(* CODESYS project ObjectOrientedProgramming(Extended).project
   Description: This example demonstrates how object orientation is used to realize a building with different rooms, which have different functions. The included visualization illustrates the implementation.
   Title: Extended Example for Object Oriented Programming

Project tree, tasks and I/O mapping:
  Device : CODESYS Control Win V3 x64, 3S - Smart Software Solutions GmbH, version 3.5.15.0
    application BuildingApplication
      libraries: Util, 3.4.1.20 (System); Standard, 3.5.15.0 (System)
      task BuildingTask (cyclic, interval t#50ms, priority 0) calls Main
      FBs/
        Light/
          function block clsDuoLight1min [ST]: ResetServiceMsg, ServiceIsNecessary, SetLifeTime
          function block clsLight1min [ST]: ServiceIsNecessary, ResetServiceMsg, SetLifeTime
          function block clsLight [ST]: Light
          function block FB_LifeTimer [ST]: Reset
        Room/
          function block clsRoom [ST]: CheckService, Operation_Nighttime, Operation_Daytime, CheckLight, ResetService, InitRoom
          function block FB_AirCondition [ST]: Reset
          function block clsClimateBetterRoom [ST]: CheckService, SetTemperature, Operation_Nighttime, Operation_Daytime, ResetService
          function block clsCheapRoom [ST]: InitRoom
          function block clsCellarRoom [ST]: InitRoom
          function block clsBetterRoom [ST]: InitRoom
      VisuElements/
        visualisation MainVisu
        visualisation PV_Room
        visualisation PV_Bulb
      program Main [ST]
      Text/
        text list TLst_OPMODE
        text list ServiceMessage
      Interfaces/
        interface IService: ServiceIsNecessary, ResetServiceMsg
        interface IRoom: Operation_Nighttime, Operation_Daytime
        interface ILight: Light
      Enums/
        data type ET_OPMODE
        data type SERVICE_MESSAGE
      license
  libraries: VisuSymbols, 3.5.10.0 (System)
  text list GlobalTextList
  00000000-0000-0000-0000-000000000000|C:\Users\m.lamp\Documents\license.txt
*)

// Device/BuildingApplication/Enums/ET_OPMODE
TYPE ET_OPMODE :
(
	NightTime := 0,
	DayTime,
	Manual
)INT;
END_TYPE

// Device/BuildingApplication/Enums/SERVICE_MESSAGE
TYPE SERVICE_MESSAGE :
(
	NO_SERVICE := 0,
	AIR_CON,
	LIGHT
	
);
END_TYPE

// Device/BuildingApplication/Main
PROGRAM Main
VAR CONSTANT
	c_iNUM_ROOM : INT := 4;
END_VAR
VAR
	CellarRoom : clsCellarRoom;
	CheapRoom : clsCheapRoom;
	BetterRoom : clsBetterRoom;   
	ClimateBetterRoom : clsClimateBetterRoom;
	
	aitfRoom : ARRAY[0..c_iNUM_ROOM - 1] OF IRoom
		:= [CellarRoom, CheapRoom, BetterRoom, ClimateBetterRoom];

(*	
	pRoom : POINTER TO clsRoom;
	xPointerValid : BOOL;
*)
	eOpMode : ET_OPMODE; 
	iSelRoom : INT;
	
	vis_iSelOpMode : INT := 0;	
	vis_sSelectDynamicText : STRING;
END_VAR

(* Initialize all of the rooms *)
CellarRoom();
CheapRoom();
BetterRoom();
ClimateBetterRoom();

(* fetch the mode: daytime, nighttime, manual *)
eOpMode := vis_iSelOpMode;
vis_sSelectDynamicText := INT_TO_STRING(eOpMode); (* text for the mode in the visu form the textlist "TLst_OPMODE"*)

FOR iSelRoom := 0 TO c_iNUM_ROOM - 1 DO
	CASE eOpMode OF
	ET_OPMODE.NightTime:
		aitfRoom[iSelRoom].Operation_Nighttime();	(* Change to night time *)
	ET_OPMODE.DayTime:
		aitfRoom[iSelRoom].Operation_Daytime(); (* Change to day time *)
	ET_OPMODE.Manual:
		;
	END_CASE	
END_FOR

END_PROGRAM

// Device/BuildingApplication/FBs/Room/clsCellarRoom
(* This room has a normal light, but no service.*)
FUNCTION_BLOCK clsCellarRoom EXTENDS clsRoom
VAR_INPUT
END_VAR
VAR_OUTPUT
END_VAR
VAR
	Light : clsLight;
END_VAR

SUPER^();
Light();

METHOD InitRoom : BOOL
VAR_INPUT
END_VAR
VAR
END_VAR
(* Asign the function block to the interface.*)
itfLight := Light;
END_METHOD

END_FUNCTION_BLOCK

// Device/BuildingApplication/FBs/Room/clsRoom
FUNCTION_BLOCK clsRoom IMPLEMENTS IRoom
VAR_INPUT
	xToggleLight : BOOL;
	xResetService : BOOL;
END_VAR
VAR_OUTPUT
	xLightON : BOOL;
	xServiceIsNecessary : BOOL;
	
END_VAR
VAR
	itfLight : ILight;	
	xInitRoom : BOOL := TRUE;
	xPrvToggleLight : BOOL;
	sServiceMessage: STRING;
END_VAR

(* Initialize the room.*)
IF xInitRoom THEN
	InitRoom();
	xInitRoom := FALSE;
END_IF

(* When the mode is set to manual, each light can be toggled. *)
IF xToggleLight AND NOT xPrvToggleLight THEN
	IF itfLight <> 0 THEN
		itfLight.Light := NOT xLightON; 
	END_IF
END_IF

(* If service is neccessary and the reset button was clicked, the service is resetted.*)
IF CheckService() <> SERVICE_MESSAGE.NO_SERVICE AND xResetService THEN
	ResetService();
END_IF

xLightON := CheckLight();

(* Convert to string, that it can be used in the visualization with the ServiceMessage text list.*)
sServiceMessage := INT_TO_STRING(CheckService());

xPrvToggleLight := xToggleLight;

METHOD CheckService : SERVICE_MESSAGE
VAR_INPUT
END_VAR
VAR
	itfService : IService;
	xItfValid : BOOL;
END_VAR
(* Check if service for the current room is neccessary. *)
IF itfLight <> 0 THEN
	xItfValid := __QUERYINTERFACE(itfLight, itfService);
	IF xItfValid THEN
		CheckService := itfService.ServiceIsNecessary;
	END_IF
END_IF
END_METHOD

METHOD Operation_Nighttime : BOOL
IF itfLight <> 0 THEN
	itfLight.Light :=TRUE;	(* Switch on the light for nighttime. *)
END_IF
END_METHOD

METHOD Operation_Daytime : BOOL
IF itfLight <> 0 THEN
	itfLight.Light := FALSE; (* No light at daytime.*)	
END_IF
END_METHOD

METHOD CheckLight : BOOL
VAR_INPUT
END_VAR
VAR
END_VAR
(* Check if the light is switched on or off.*)
IF itfLight <> 0 THEN
	CheckLight := itfLight.Light;
END_IF
END_METHOD

METHOD ResetService : BOOL
VAR_INPUT
END_VAR
VAR
	itfService : IService;
	xItfValid : BOOL;
END_VAR
(* Resets the service for one room. *)
IF itfLight <> 0 THEN
	xItfValid := __QUERYINTERFACE(itfLight, itfService);
	IF xItfValid THEN
		ResetService := itfService.ResetServiceMsg();
	END_IF
END_IF
END_METHOD

(* Initialize the room.*)
METHOD InitRoom : BOOL
VAR_INPUT
END_VAR
VAR
END_VAR
(* This method is empty, but overriden from the function block, which inherit this
function block.*)
END_METHOD

END_FUNCTION_BLOCK

// Device/BuildingApplication/Interfaces/IRoom
(* Interface for a room.*)
INTERFACE IRoom EXTENDS __System.IQueryInterface

METHOD Operation_Nighttime : BOOL
VAR_INPUT
END_VAR
VAR
END_VAR
END_METHOD

METHOD Operation_Daytime : BOOL
VAR_INPUT
END_VAR
VAR
END_VAR
END_METHOD

END_INTERFACE

// Device/BuildingApplication/Interfaces/ILight
(* Interface for a light bulb. *)
INTERFACE ILight EXTENDS __System.IQueryInterface

PROPERTY Light : BOOL
SET
END_SET
GET
END_GET
END_PROPERTY

END_INTERFACE

// Device/BuildingApplication/Interfaces/IService
(* Interface for the service.*)
INTERFACE IService EXTENDS __System.IQueryInterface

PROPERTY ServiceIsNecessary : SERVICE_MESSAGE
GET
END_GET
END_PROPERTY

METHOD ResetServiceMsg : BOOL
VAR_INPUT
END_VAR
VAR
END_VAR
END_METHOD

END_INTERFACE

// Device/BuildingApplication/FBs/Light/clsLight
FUNCTION_BLOCK clsLight IMPLEMENTS ILight
VAR_INPUT
	xOnOff : BOOL; (* If TRUE, the light is enabled *)
END_VAR
VAR_OUTPUT
	xValue : BOOL; (* If True, the light is enabled.*)
END_VAR
VAR
	RT_OnOff : R_TRIG;
	FT_OnOff : F_TRIG;
END_VAR

(* True, if rising edge --> light is switched on*)
RT_OnOff(CLK:= xOnOff);
IF RT_OnOff.Q THEN
	xValue := TRUE;
END_IF

(* True, if falling edge --> light is switched off *)
FT_OnOff(CLK:= xOnOff);
IF FT_OnOff.Q THEN
	xValue := FALSE;
END_IF

PROPERTY Light : BOOL
GET
(* True, when the light is switched on *)
Light := xValue;
END_GET
SET
(* Set to true, when the light is switched on.*)
xValue := Light;
END_SET
END_PROPERTY

END_FUNCTION_BLOCK

// Device/BuildingApplication/FBs/Room/clsCheapRoom
(* This room has a normal light and a service.*)
FUNCTION_BLOCK clsCheapRoom EXTENDS clsRoom
VAR_INPUT
END_VAR
VAR_OUTPUT
END_VAR
VAR
	Light1min : clsLight1min;
END_VAR

SUPER^();
Light1min();

METHOD InitRoom : BOOL
VAR_INPUT
END_VAR
VAR
END_VAR
(* Asign the function block to the interface.*)
itfLight := Light1min;
END_METHOD

END_FUNCTION_BLOCK

// Device/BuildingApplication/FBs/Light/clsLight1min
FUNCTION_BLOCK clsLight1min EXTENDS clsLight IMPLEMENTS IService
VAR_INPUT
	xNewLight : BOOL;
END_VAR
VAR_OUTPUT
	xPleaseInsertNewLight : BOOL;
	eServiceMessage : SERVICE_MESSAGE;
END_VAR
VAR
	xInitLifeTimer : BOOL := TRUE;
	LifeTimer : FB_LifeTimer;
END_VAR

(* call the clsLight function block *)
SUPER^();

(* Initialize the lifetime of the light bulb *)
IF xInitLifeTimer THEN
	SetLifeTime(); (* set time for LifeTimer *)
	xInitLifeTimer := FALSE;
END_IF

(* Count down the life time, if xNewLight is True, the lifetime is resetted.*)
LifeTimer(xOnOff:= xValue, xReset:= xNewLight);

(* If the end of the liftime is reached, a service message is generated.*)
IF LifeTimer.xAlive THEN
	eServiceMessage := SERVICE_MESSAGE.NO_SERVICE;
ELSE
	eServiceMessage := SERVICE_MESSAGE.LIGHT;
END_IF

PROPERTY ServiceIsNecessary : SERVICE_MESSAGE
GET
(* Return the service Message.*)
ServiceIsNecessary := eServiceMessage;
END_GET
END_PROPERTY

METHOD ResetServiceMsg : BOOL
VAR_INPUT
END_VAR
VAR
END_VAR
(* Reset the lifetime of the light. *)
IF eServiceMessage <> SERVICE_MESSAGE.NO_SERVICE THEN
	LifeTimer.Reset();	
END_IF
END_METHOD

METHOD SetLifeTime : BOOL
VAR_INPUT
END_VAR
VAR
END_VAR
(* Set the lifetime of the light bulb in minutes.*)
LifeTimer.iTime := 1;
END_METHOD

END_FUNCTION_BLOCK

// Device/BuildingApplication/FBs/Light/FB_LifeTimer
FUNCTION_BLOCK FB_LifeTimer
VAR_INPUT
	xOnOff : BOOL; (* True when the light is enabled *)
	xReset : BOOL;
	iTime : INT; (* Lifetime in minutes *)
END_VAR
VAR_OUTPUT
	xAlive : BOOL; (* True, when the life time is countedn down to zero.*)
	iRemainingTime : INT; (* remaining lifetime of the light in minutes.*)
END_VAR
VAR
	xInit : BOOL := TRUE;
	iSeconds : INT := 0;
	ton1SecTriggerSignal : TON; (* Timer for couting the seconds *)
END_VAR

(* Initialize the life time of the light.*)
IF xInit THEN
	iRemainingTime := iTime; (* time in minutes *)
	xInit := FALSE;
END_IF

(* After 1 second the In value is switched and the timer is started again, when the light is
switched on.*)
ton1SecTriggerSignal(IN:= xOnOff AND NOT ton1SecTriggerSignal.Q AND xAlive AND NOT xReset, 
					 PT:= T#1000MS);

(* After one second, one second is decrement.*)
IF ton1SecTriggerSignal.Q THEN
	IF iSeconds < 60 THEN
		iSeconds := iSeconds + 1; (* Count the seconds.*)
	ELSE
		(* Remeining time in minutes *)
		iRemainingTime := iRemainingTime - 1;
		iSeconds := 0;
	END_IF
END_IF

(* Be pressing the reset button, the original lifetime is set.*)
IF xReset THEN
	iRemainingTime := iTime;
	iSeconds := 0;
END_IF

(* Check if the end of the lifetime is reached or not. *)
xAlive := NOT (iRemainingTime <= 0);

METHOD Reset : BOOL
VAR_INPUT
END_VAR
VAR
END_VAR
(* Reset the timer. *)
iRemainingTime := iTime;
iSeconds := 0;
END_METHOD

END_FUNCTION_BLOCK

// Device/BuildingApplication/FBs/Room/clsBetterRoom
(* This room has a duo light. Has a doubled lifetime from a normal one.*)
FUNCTION_BLOCK clsBetterRoom EXTENDS clsRoom
VAR_INPUT
END_VAR
VAR_OUTPUT
END_VAR
VAR
	DuoLight1min : clsDuoLight1min;
END_VAR

(* Call the clsRoom function block. *)
SUPER^();
(* Initialize the lifetime for the light bulb.*)
DuoLight1min();

METHOD InitRoom : BOOL
VAR_INPUT
END_VAR
VAR
END_VAR
(* Asign the function block to the interface.*)
itfLight := DuoLight1min;
END_METHOD

END_FUNCTION_BLOCK

// Device/BuildingApplication/FBs/Light/clsDuoLight1min
FUNCTION_BLOCK clsDuoLight1min EXTENDS clsLight1min
VAR_INPUT
	xNewSecondLight : BOOL;
END_VAR
VAR_OUTPUT
	xSecondValue : BOOL;
	xPleaseInsertNewSecondLight : BOOL;
END_VAR
VAR
	SecondLifeTimer : FB_LifeTimer;
END_VAR

SUPER^(); (* start the First Lifetimer and call SetLifeTime Method. The method
			from this function block is used, because it has overridden the other one.*)

(* Start the second life timer *)
IF NOT LifeTimer.xAlive THEN
	SecondLifeTimer(xOnOff:= xSecondValue, xReset:= xNewSecondLight);
END_IF

(* When the lifetimer has counted down to zero, a new light has to be inserted.*)
IF NOT LifeTimer.xAlive AND NOT SecondLifeTimer.xAlive AND SecondLifeTimer.iRemainingTime = 0 THEN
	eServiceMessage := SERVICE_MESSAGE.LIGHT;
ELSE
	eServiceMessage := SERVICE_MESSAGE.NO_SERVICE;
END_IF

(* If xValue = TRUE the light was switched on, if FALSE then the light was switched off*)
xSecondValue := xValue;

METHOD ResetServiceMsg : BOOL
VAR_INPUT
END_VAR
VAR
END_VAR
(* Reset the lifetime of the first timer for the light. *)
SUPER^.ResetServiceMsg();
(* Reset the lifetime of the second timer for the light*)
IF eServiceMessage <> SERVICE_MESSAGE.NO_SERVICE THEN
	SecondLifeTimer.Reset();	
END_IF
END_METHOD

PROPERTY ServiceIsNecessary : SERVICE_MESSAGE
GET
(* Service is neccessary when both timer have reached the end, then the service message is set.*)
ServiceIsNecessary := eServiceMessage;
END_GET
END_PROPERTY

METHOD SetLifeTime : BOOL
VAR_INPUT
END_VAR
VAR
END_VAR
(* set the lifetime of the light bulb in minutes *)
SUPER^.SetLifeTime();
(* set the second lifetime of the light bulb in minutes, because it is a duo light. *)
SecondLifeTimer.iTime := 1;
END_METHOD

END_FUNCTION_BLOCK

// Device/BuildingApplication/FBs/Room/clsClimateBetterRoom
(* This room has a duo light and an air condition, for regulating the temperature for
daytime and nighttime. *)
FUNCTION_BLOCK clsClimateBetterRoom EXTENDS clsBetterRoom
VAR_INPUT
	
END_VAR
VAR_OUTPUT
END_VAR
VAR
	AirCondition : FB_AirCondition; (* Air condition, which regulates the temperature. *)
	xChangeAirConditionFilter : BOOL; (* After a certain time, the filter has to bec changed.*)
	iActTemp : INT; (* The current temperature.*)
END_VAR

SUPER^();

(* Regulate the temperatur.*)
AirCondition( iActTemp=> iActTemp);

(* After a certain amount of changes from day- and nighttime, the filter has to bec changed.*)
IF AirCondition.iCounter > 5 THEN
	xChangeAirConditionFilter := TRUE;
ELSE
	xChangeAirConditionFilter := FALSE;
END_IF

METHOD CheckService : SERVICE_MESSAGE
VAR_INPUT
END_VAR
VAR
	itfService : IService;
	xItfValid : BOOL;
END_VAR
(* Check the service for the room.*)
CheckService := SERVICE_MESSAGE.NO_SERVICE;

IF  SUPER^.CheckService() <> SERVICE_MESSAGE.NO_SERVICE THEN
	CheckService := SUPER^.CheckService(); (* Service for the light bulb.*)
ELSIF xChangeAirConditionFilter THEN
	CheckService := SERVICE_MESSAGE.AIR_CON; (* service for the air condition. *)
END_IF
END_METHOD

METHOD SetTemperature : INT
VAR_INPUT
	iValue : INT;
END_VAR
VAR
END_VAR
(* Set the current temperature.*)
AirCondition.iSetTemp := iValue;
END_METHOD

METHOD Operation_Nighttime : BOOL
SUPER^.Operation_Nighttime(); (* switch on the light.*)
SetTemperature(15); (*Set the temperature for the night time. *)
END_METHOD

METHOD Operation_Daytime : BOOL
SUPER^.Operation_Daytime(); (* switch off the light.*)
SetTemperature(21); (* Set temperature for daytime *)
END_METHOD

METHOD ResetService : BOOL
VAR
	itfService : IService;
	xItfValid : BOOL;
END_VAR
IF xChangeAirConditionFilter THEN
	AirCondition.Reset(); (* Reset the air contition.*)
ELSE
	SUPER^.ResetService(); (* Reset the light. *)
END_IF
END_METHOD

END_FUNCTION_BLOCK

// Device/BuildingApplication/FBs/Room/FB_AirCondition
FUNCTION_BLOCK FB_AirCondition
VAR_INPUT
	iSetTemp : INT;
END_VAR
VAR_OUTPUT
	iActTemp : INT;
	iCounter : INT;
END_VAR
VAR
	iSetCmp : INT;
	TempController : RAMP_INT;
END_VAR

(* If the temperature has changed, the counter is increased by one.
	At a certain value, the filter for the air con has to be changed.*)
IF iSetCmp <> iSetTemp THEN
	iCounter := iCounter + 1;
END_IF

(* Set the value to compare to the new value.*)
iSetCmp := iSetTemp;

TempController(IN:= iSetTemp, ASCEND:= 20, DESCEND:= 10, TIMEBASE:= T#5S, 
		       OUT=> iActTemp);

METHOD Reset
VAR_INPUT
END_VAR
(* Reset the counter for a new filter. *)
iCounter := 0;
END_METHOD

END_FUNCTION_BLOCK

// Device/BuildingApplication/VisuElements/MainVisu
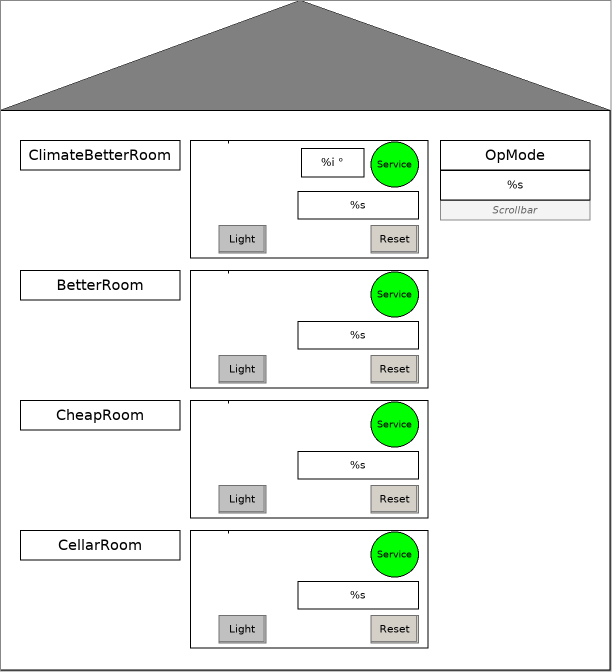
VISUALIZATION MainVisu  // 612x672
    Rectangle (0,110 610x560)
    Frame (190,140 240x120)
        shows PV_Room(Room := Main.ClimateBetterRoom)
        p218911849: Main.ClimateBetterRoom
    Frame (190,530 240x120)
        shows PV_Room(Room := Main.CellarRoom)
        p218911849: Main.CellarRoom
    Frame (190,400 240x120)
        shows PV_Room(Room := Main.CheapRoom)
        p218911849: Main.CheapRoom
    Frame (190,270 240x120)
        shows PV_Room(Room := Main.BetterRoom)
        p218911849: Main.BetterRoom
    Scrollbar (440,200 150x20)
        p1057716461: Main.vis_iSelOpMode
    Rectangle (440,170 150x30), "%s", text list: 'TLst_OPMODE', text index: Main.vis_sSelectDynamicText
    Rectangle (440,140 150x30), "OpMode"
    Polygon (300,0) (610,110) (0,110)
    Rectangle (20,140 160x30), "ClimateBetterRoom"
    Rectangle (20,270 160x30), "BetterRoom"
    Rectangle (20,400 160x30), "CheapRoom"
    Rectangle (20,530 160x30), "CellarRoom"
    Rectangle (301,148 63x29), "%i °", text variable: Main.ClimateBetterRoom.iActTemp
END_VISUALIZATION

// Device/BuildingApplication/VisuElements/PV_Room
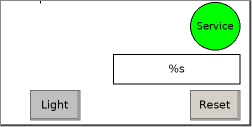
VISUALIZATION PV_Room  // 252x127
VAR_IN_OUT
	Room : clsRoom;
END_VAR
    Rectangle (0,0 250x125)
    Frame (40,0 30x50)
        shows PV_Bulb(xValue := Room.xLightON)
    Ellipse (190,2 50x48), "Service", colour toggle: Room.sServiceMessage <> '0'
    Button (190,90 50x30), "Reset"
        tap Room.xResetService
    Button (30,90 50x30), "Light", colour toggle: Room.xToggleLight
        tap Room.xToggleLight
    Rectangle (113,54 127x30), "%s", text list: 'ServiceMessage', text index: Room.sServiceMessage
END_VISUALIZATION

// Device/BuildingApplication/VisuElements/PV_Bulb
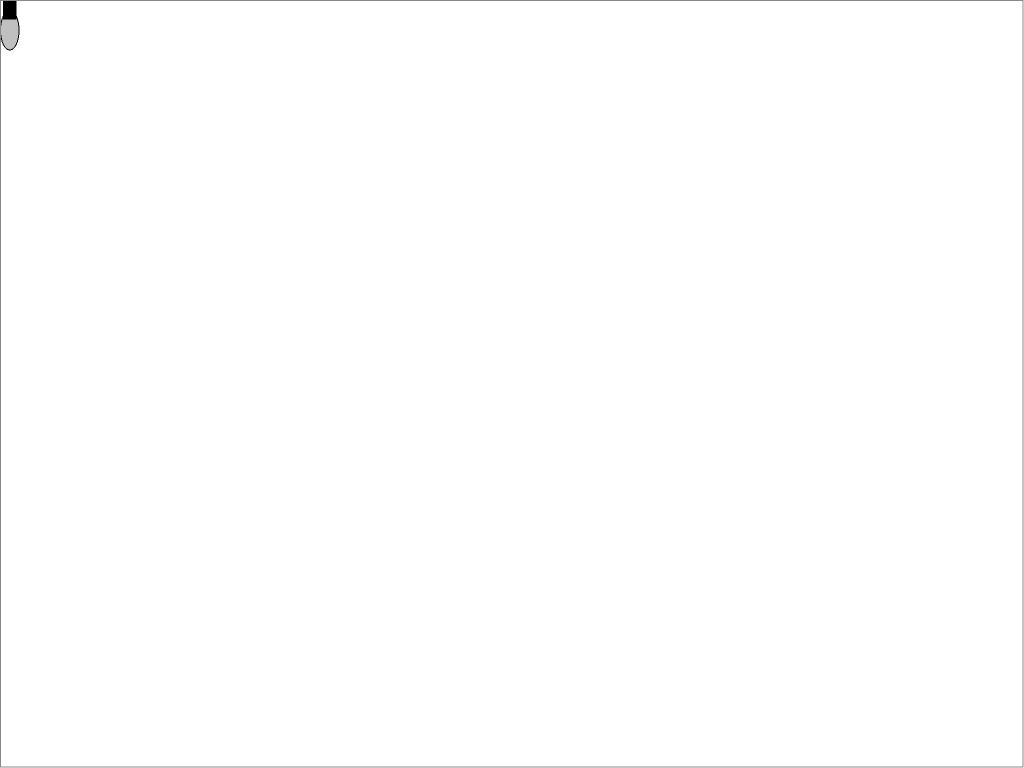
VISUALIZATION PV_Bulb  // 1024x768
VAR_INPUT
	xValue : BOOL;
END_VAR
    Ellipse (0,10 19x40), colour toggle: xValue
    Rectangle (3,0 13x19)
END_VISUALIZATION

(* text list TLst_OPMODE (id | default)
  0 | NightTime
  1 | DayTime
  2 | Manual
   |  *)

(* text list ServiceMessage (id | default)
  0 | No Service.
  1 | New filter.
  2 | New light.
   |  *)
